// TIA Portal V18 export
TYPE "UDT_Marking StringToChar"
// stored: IsFailsafeCompliant false
   STRUCT
      "Char" : Array[0..127] of Char;
   END_STRUCT;
END_TYPE
